{attribute addProperty BoxType "EK1122-0000-0018"}
{attribute addProperty Id "Beckhoff_EL32xxsub_EK1100EK1100_179A0949162"}
{attribute addProperty CRC "2445542956"}
{attribute addProperty SizeInBites "16"}
{attribute addProperty SizeInBytes "2"}
TYPE Beckhoff_EL32xxEK1122_91C4062C EXTENDS EK1122_179A0949 :
STRUCT
	{attribute addProperty Name "Beckhoff_EL32xxsub_EK1100"}
	Beckhoff_EL32xxsub_EK1100 : EK1100_179A0949;
END_STRUCT
END_TYPE

(* stored: Version 1.2.0.0, ProductVersion 3.1.4024.9
   DUT Beckhoff_EL32xxEK1122_91C4062C: Id {03216c9c-162d-4ec4-8c69-20bd112ec447} *)
